(* IEC 61131-3 sources: CodesysTest/alpha/export/FBs/Components/Cylinders/FB_ThreePositionCylinder.pou, 1 file *)

(* ---- ExtendCylinderLowPressure.m.st ---- *)
(*#-#-#-#-#-#-#-#-#-#---Declaration---#-#-#-#-#-#-#-#-#-#-#-#-#*)

METHOD ExtendCylinderLowPressure
VAR_INPUT
END_VAR
(*#-#-#-#-#-#-#-#-#-#---Implementation---#-#-#-#-#-#-#-#-#-#-#-#-#*)

extendOutput := TRUE;
retractOutput := TRUE;
